{attribute addProperty BoxType "EK1100-0000-0018"}
{attribute addProperty Id "Beckhoff_EK18xxEK1122Beckhoff_EK18xxEK1122_46BB19D81271158.875"}
{attribute addProperty CRC "733156242"}
{attribute addProperty SizeInBites "1271"}
{attribute addProperty SizeInBytes "158.875"}
TYPE Beckhoff_EK18xx_2BB31392 EXTENDS EK1100_179A0949 :
STRUCT
	{attribute addProperty Name "Beckhoff_EK18xxEK1122"}
	Beckhoff_EK18xxEK1122 : Beckhoff_EK18xxEK1122_46BB19D8;
END_STRUCT
END_TYPE

(* stored: Version 1.2.0.0, ProductVersion 3.1.4024.9
   DUT Beckhoff_EK18xx_2BB31392: Id {b590e900-3878-43aa-86db-6c57528e4cc5} *)
